PROGRAM MAIN
VAR
	fbKL6581			: FB_KL6581;

	fbRec_RPS_Switch	: FB_Rec_RPS_Switch;
	dwId				: DWORD := 1059793;
	stEnOceanSwitch		: STR_EnOceanSwitch;
	bReady				: BOOL;
	bBusy				: BOOL;
	bError				: BOOL;
	iErrorId			: INT;
END_VAR

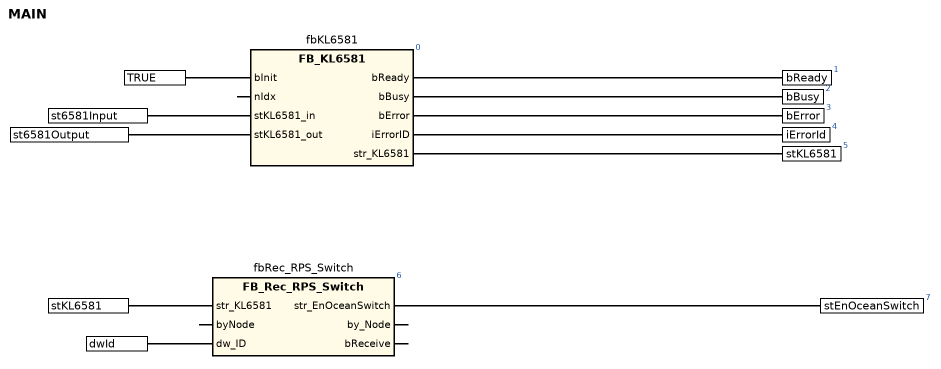
fbKL6581(bInit := TRUE, stKL6581_in := st6581Input, stKL6581_out := st6581Output); // FB_KL6581
bReady := fbKL6581.bReady;
bBusy := fbKL6581.bBusy;
bError := fbKL6581.bError;
iErrorId := fbKL6581.iErrorID;
stKL6581 := fbKL6581.str_KL6581;
fbRec_RPS_Switch(str_KL6581 := stKL6581, dw_ID := dwId); // FB_Rec_RPS_Switch
stEnOceanSwitch := fbRec_RPS_Switch.str_EnOceanSwitch;

END_PROGRAM

(* stored: Version 1.1.0.1, ProductVersion 3.1.4022.10
   POU MAIN: Id {d8c5785e-b7a4-4a76-a9e7-c4771294d345}, SpecialFunc None *)
